{attribute 'GeneratedUsingTerminal: EP2339-0042-0017'}
{attribute addProperty BoxType "EP2339-0042-0017"}
{attribute addProperty Id "OutputAT %Q*BOOL1"}
{attribute addProperty CRC "1120571895"}
{attribute addProperty Size "1"}
TYPE DO_X04_Pin_42CA91F7 EXTENDS OutputBase_10CEE7DE :
STRUCT
	{attribute addProperty Name "Output"}
	Output AT %Q* : BOOL;
END_STRUCT
END_TYPE

(* stored: Version 1.2.0.0, ProductVersion 3.1.4024.11
   DUT DO_X04_Pin_42CA91F7: Id {3dc327fe-2ed7-456d-89ad-6b4d86879d3d} *)
